# EPICS substitutions: RadiationMonitoringApp/Db/site/peripheral-station.substitutions
file ecogamma.template{
     pattern {LOCA,UNIT,PORT }
             {SITE,$(UNIT),$(GPORT)}
}

#file fht40G.template{
#     pattern {P,PORT,N,M}
#             {RADM:SITE:$(UNIT),$(NPORT),0,0}
#}
